// TIA Portal project "babu_CounterConveyor" (V15)

(* hardware
DEVICE "S7-1200 station_1"  S7-1200 Station
   slot 0: "Rack_0"  S7-1200 Rack  Rack  V1.0
   slot 1: "PLC_1"  CPU 1212C DC/DC/DC  6ES7 212-1AE40-0XB0  V4.2
*)

// ===== PLC "PLC_1"  CPU 1212C DC/DC/DC =====

VAR_GLOBAL   // PLC tag table "Default tag table"
   "PUSH BUTTON" AT %M0.0 : Bool;
   "PUSH BUTTON MEMORY" AT %M0.1 : Bool;
   "PULSE" AT %M0.2 : Bool;
   "PULSE ON" AT %M0.3 : Bool;
   "Fill Bottle MEM" AT %M0.4 : Bool;
   "Fill Bottle" AT %Q0.0 : Bool;
   "Conveyor" AT %Q0.1 : Bool;
   "BOTTLE SENSOR" AT %M0.5 : Bool;
   "COMPLETED" AT %Q0.2 : Bool;
END_VAR

// folder: System blocks/Program resources

DATA_BLOCK "IEC_Timer_0_DB"   // DB1
{ S7_Optimized_Access := 'TRUE' }
AUTHOR : Simatic
FAMILY : IEC
NAME : IEC_TMR
VERSION : 1.0
// stored: InstanceOfName IEC_TIMER
"IEC_TIMER"
BEGIN
END_DATA_BLOCK

DATA_BLOCK "IEC_Timer_0_DB_1"   // DB2
{ S7_Optimized_Access := 'TRUE' }
AUTHOR : Simatic
FAMILY : IEC
NAME : IEC_TMR
VERSION : 1.0
// stored: InstanceOfName IEC_TIMER
"IEC_TIMER"
BEGIN
END_DATA_BLOCK

DATA_BLOCK "IEC_Timer_0_DB_2"   // DB3
{ S7_Optimized_Access := 'TRUE' }
AUTHOR : Simatic
FAMILY : IEC
NAME : IEC_TMR
VERSION : 1.0
// stored: InstanceOfName IEC_TIMER
"IEC_TIMER"
BEGIN
END_DATA_BLOCK

DATA_BLOCK "IEC_Timer_0_DB_3"   // DB4
{ S7_Optimized_Access := 'TRUE' }
AUTHOR : Simatic
FAMILY : IEC
NAME : IEC_TMR
VERSION : 1.0
// stored: InstanceOfName IEC_TIMER
"IEC_TIMER"
BEGIN
END_DATA_BLOCK

DATA_BLOCK "IEC_Timer_0_DB_4"   // DB5
{ S7_Optimized_Access := 'TRUE' }
AUTHOR : Simatic
FAMILY : IEC
NAME : IEC_TMR
VERSION : 1.0
// stored: InstanceOfName IEC_TIMER
"IEC_TIMER"
BEGIN
END_DATA_BLOCK

DATA_BLOCK "IEC_Timer_0_DB_6"   // DB8
{ S7_Optimized_Access := 'TRUE' }
AUTHOR : Simatic
FAMILY : IEC
NAME : IEC_TMR
VERSION : 1.0
// stored: InstanceOfName IEC_TIMER
"IEC_TIMER"
BEGIN
END_DATA_BLOCK

DATA_BLOCK "IEC_Counter_0_DB_1"   // DB9
{ S7_Optimized_Access := 'TRUE' }
AUTHOR : Simatic
FAMILY : IEC
NAME : CNTR
VERSION : 1.0
// stored: InstanceOfName IEC_COUNTER
"IEC_COUNTER"
BEGIN
END_DATA_BLOCK

// folder: (top level)

ORGANIZATION_BLOCK "Main"   // OB1, LAD, ProgramCycle
TITLE = "Main Program Sweep (Cycle)"
{ S7_Optimized_Access := 'TRUE' }
VERSION : 0.1
   VAR_INPUT
      Initial_Call : Bool;   // Initial call of this OB
      Remanence : Bool;   // =True, if remanent data are available
   END_VAR
   VAR_TEMP   // added for the SCL form of the ladder/FBD networks
      _w1 : Bool;
   END_VAR
BEGIN

REGION Network 1
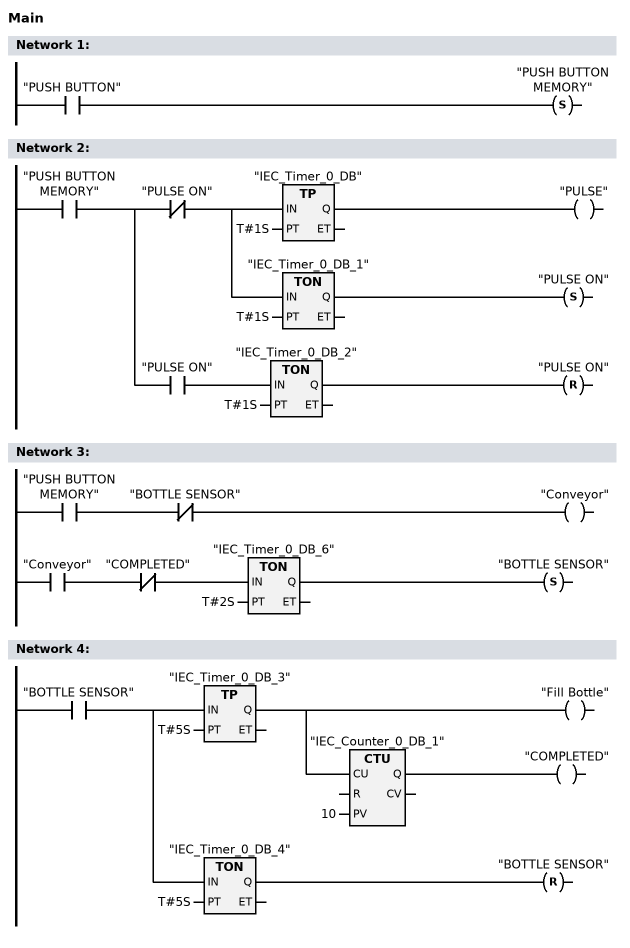
   RUNG wire#powerrail
      Contact( "PUSH BUTTON" )
      S_Coil( "PUSH BUTTON MEMORY" )
   END_RUNG
   // the same network as SCL:
   IF "PUSH BUTTON" THEN "PUSH BUTTON MEMORY" := TRUE; END_IF;
END_REGION

REGION Network 2
   #_w1 := "PUSH BUTTON MEMORY" AND NOT "PULSE ON";
   "IEC_Timer_0_DB".TP(IN := #_w1, PT := T#1S);
   "PULSE" := "IEC_Timer_0_DB".Q;
   "IEC_Timer_0_DB_1".TON(IN := #_w1, PT := T#1S);
   IF "IEC_Timer_0_DB_1".Q THEN "PULSE ON" := TRUE; END_IF;
   "IEC_Timer_0_DB_2".TON(IN := "PUSH BUTTON MEMORY" AND "PULSE ON", PT := T#1S);
   IF "IEC_Timer_0_DB_2".Q THEN "PULSE ON" := FALSE; END_IF;
END_REGION

REGION Network 3
   "Conveyor" := "PUSH BUTTON MEMORY" AND NOT "BOTTLE SENSOR";
   "IEC_Timer_0_DB_6".TON(IN := "Conveyor" AND NOT "COMPLETED", PT := T#2S);
   IF "IEC_Timer_0_DB_6".Q THEN "BOTTLE SENSOR" := TRUE; END_IF;
END_REGION

REGION Network 4
   "IEC_Timer_0_DB_3".TP(IN := "BOTTLE SENSOR", PT := T#5S);
   "Fill Bottle" := "IEC_Timer_0_DB_3".Q;
   "IEC_Counter_0_DB_1".CTU(CU := "IEC_Timer_0_DB_3".Q, PV := 10);
   "COMPLETED" := "IEC_Counter_0_DB_1".Q;
   "IEC_Timer_0_DB_4".TON(IN := "BOTTLE SENSOR", PT := T#5S);
   IF "IEC_Timer_0_DB_4".Q THEN "BOTTLE SENSOR" := FALSE; END_IF;
END_REGION
END_ORGANIZATION_BLOCK